FUNCTION_BLOCK AsyncManager
VAR
	asyncResponses : Dictionary;
	config : I_AsyncManagerConfig;
END_VAR

METHOD PUBLIC ConvertResponseToAsync
VAR_INPUT
	Response : I_ServerResponse;
	AsyncResponse : REFERENCE TO I_ServerResponse;
END_VAR
VAR
	sessionId : T_MAXSTRING;
	newResponse : I_ServerResponse;
END_VAR
IF NOT config.TryGetSessionIdFromResponse(Response,sessionId) THEN
	Response.Error('Failed to convert response to async-response, missing Session Id');
	RETURN;
END_IF

IF AsyncResponse <> 0 THEN
	AsyncResponse.Error('Response has been replaced');
END_IF

//AsyncResponse := Response.Clone(
END_METHOD

METHOD FB_init : BOOL
VAR_INPUT
	bInitRetains : BOOL; // if TRUE, the retain variables are initialized (warm start / cold start)
	bInCopyCode : BOOL;  // if TRUE, the instance afterwards gets moved into the copy code (online change)
	Config : I_AsyncManagerConfig;
END_VAR
THIS^.config := Config;
END_METHOD

END_FUNCTION_BLOCK

(* stored: Version 1.1.0.1, ProductVersion 3.1.4024.12
   POU AsyncManager: Id {3f208033-fc55-4901-a839-41a96f923931}, SpecialFunc None
   Folder Constructor: Id {4cf791e2-033e-41c1-bd7f-0547acd5686e}
   Method ConvertResponseToAsync: Id {4f8caf87-0ff4-4c38-a46f-c7cc9de3a703}
   Method FB_init: Id {53fea6ea-86b0-4213-974d-53d7704695f3} *)
